// TIA Portal V16 export
// export: Created 2022-11-01T21:54:09.9241492Z, ExportSetting WithDefaults, DisplayName Totally Integrated Automation Portal, DisplayVersion V16, DisplayName TIA Portal Version Control Interface, DisplayVersion V16, DisplayName TIA Portal Openness, DisplayVersion V16, DisplayName SINAMICS Startdrive Advanced, DisplayVersion V16, DisplayName SINAMICS Startdrive G130, G150, S120, S150, SINAMICS MV, S210, DisplayVersion V16, DisplayName SINAMICS Startdrive G110M, G120, G120C, G120D, G120P, DisplayVersion V16, DisplayName STEP 7 Professional, DisplayVersion V16, DisplayName STEP 7 Safety, DisplayVersion V16, DisplayName WinCC Professional, DisplayVersion V16
VAR_GLOBAL   // PLC tag table "AI C700"
   iTIR701 AT %IW1300 : Int;
   iTIR702 AT %IW1302 : Int;
   iTIR703 AT %IW1304 : Int;
   iTIR704 AT %IW1306 : Int;
   iTIR705 AT %IW1308 : Int;
   iTIR706 AT %IW1310 : Int;
   iTIR707 AT %IW1312 : Int;
   iTIR708 AT %IW1314 : Int;
   iTIR709 AT %IW1316 : Int;
   iTIR710 AT %IW1318 : Int;
   iTIR711 AT %IW1320 : Int;
   iTIR712 AT %IW1322 : Int;
   iTIR713 AT %IW1324 : Int;
   iTIR714 AT %IW1326 : Int;
   iTIR715 AT %IW1328 : Int;
   iTIR716 AT %IW1330 : Int;
   iTIR717 AT %IW1332 : Int;
   iTIR718 AT %IW1334 : Int;
   iTIR719 AT %IW1336 : Int;
   iTIR720 AT %IW1338 : Int;
   iTIR721 AT %IW1340 : Int;
   iTIR722 AT %IW1342 : Int;
   iTIR723 AT %IW1344 : Int;
   iTIR724 AT %IW1346 : Int;
   iTIR725 AT %IW1348 : Int;
   iTIR726 AT %IW1350 : Int;
   iTIR727 AT %IW1352 : Int;
   iTIR728 AT %IW1354 : Int;
   iTIR729 AT %IW1356 : Int;
   iTIR730 AT %IW1358 : Int;
   iTIR731 AT %IW1360 : Int;
   iTIR732 AT %IW1362 : Int;
   iTIR733 AT %IW1364 : Int;
   iTIR734 AT %IW1366 : Int;
   iTIR735 AT %IW1368 : Int;
   iTIR736 AT %IW1370 : Int;
   iTIR737 AT %IW1372 : Int;
   iTIR738 AT %IW1374 : Int;
   iTIR739 AT %IW1376 : Int;
   iTIR740 AT %IW1378 : Int;
   iTIR741 AT %IW1380 : Int;
   iTIR742 AT %IW1382 : Int;
   iTIR743 AT %IW1384 : Int;
   iTIR744 AT %IW1386 : Int;
   iTIR745 AT %IW1388 : Int;
   iTIR746 AT %IW1390 : Int;
   iTIR747 AT %IW1392 : Int;
   iTIR748 AT %IW1394 : Int;
   iTIR749 AT %IW1396 : Int;
   iTIR750 AT %IW1398 : Int;
   iTIR751 AT %IW1400 : Int;
   iTIR752 AT %IW1402 : Int;
   iTIR753 AT %IW1404 : Int;
   iTIR754 AT %IW1406 : Int;
   iTIR755 AT %IW1408 : Int;
   iTIR756 AT %IW1410 : Int;
   iTIR757 AT %IW1412 : Int;
   iTIR758 AT %IW1414 : Int;
   iTIR759 AT %IW1416 : Int;
   iTIR760 AT %IW1418 : Int;
   iTIR761 AT %IW1420 : Int;
   iTIR762 AT %IW1422 : Int;
   iQIR701 AT %IW1424 : Int;
   iQIR702 AT %IW1426 : Int;
   iQIR703 AT %IW1428 : Int;
   iQIR704 AT %IW1430 : Int;
   iPIR701 AT %IW1432 : Int;
   iPIR702 AT %IW1434 : Int;
   iPIR703 AT %IW1436 : Int;
   iPIR704 AT %IW1438 : Int;
   iPIR705 AT %IW1440 : Int;
   iPIR706 AT %IW1442 : Int;
   iPIR707 AT %IW1444 : Int;
   iPIR708 AT %IW1446 : Int;
   iPIR709 AT %IW1448 : Int;
   iPIR710 AT %IW1450 : Int;
   iPIR711 AT %IW1452 : Int;
   iPIR712 AT %IW1454 : Int;
   iPIR713_virtual AT %IW1456 : Int;
   iPIR714 AT %IW1458 : Int;
   iPIR715 AT %IW1460 : Int;
   iPIR716_virtual AT %IW1462 : Int;
   iPIR717 AT %IW1464 : Int;
   iPIR718 AT %IW1466 : Int;
   iPIR719_virtual AT %IW1468 : Int;
   iPIR720 AT %IW1470 : Int;
   iPIR721 AT %IW1472 : Int;
   iPIR722 AT %IW1474 : Int;
   iPIR723 AT %IW1476 : Int;
   iPIR724 AT %IW1478 : Int;
   iPIR725 AT %IW1480 : Int;
   iPIR726 AT %IW1482 : Int;
   iPIR727 AT %IW1484 : Int;
   iPIR728 AT %IW1486 : Int;
   iLIR701 AT %IW1488 : Int;
   iLIR702 AT %IW1490 : Int;
   iLIR703 AT %IW1492 : Int;
   iLIR704 AT %IW1494 : Int;
   iLIR705 AT %IW1496 : Int;
   iLIR706 AT %IW1498 : Int;
   iLIR707 AT %IW1500 : Int;
   iLIR708 AT %IW1502 : Int;
   iLIR709 AT %IW1504 : Int;
   iLIR710 AT %IW1506 : Int;
   iLIR711 AT %IW1508 : Int;
   iLIR712 AT %IW1510 : Int;
   iLIR713 AT %IW1512 : Int;
   iLIR714 AT %IW1514 : Int;
   iLIR715 AT %IW1516 : Int;
   iLIR716 AT %IW1518 : Int;
   iLIR717 AT %IW1520 : Int;
   iLIR718 AT %IW1522 : Int;
   iLIR719 AT %IW1524 : Int;
   iLIR720 AT %IW1526 : Int;
   iLIR721 AT %IW1528 : Int;
   iFIR701 AT %IW1530 : Int;
   iFIR702 AT %IW1532 : Int;
   iFIR703 AT %IW1534 : Int;
   iFIR704 AT %IW1536 : Int;
   iFIR705 AT %IW1538 : Int;
   iFIR706 AT %IW1540 : Int;
   iFIR707 AT %IW1542 : Int;
   iFIR708 AT %IW1544 : Int;
   iFIR709 AT %IW1546 : Int;
   iFIR710 AT %IW1548 : Int;
   iFIR711 AT %IW1550 : Int;
   iFIR712 AT %IW1552 : Int;
   iFIR713 AT %IW1554 : Int;
   iFIR714 AT %IW1556 : Int;
   iFIR715 AT %IW1558 : Int;
   iFIR716 AT %IW1560 : Int;
   iFIR717 AT %IW1562 : Int;
   iFIR718 AT %IW1564 : Int;
   iFIR719 AT %IW1566 : Int;
   iFIR720 AT %IW1568 : Int;
   iFIR721 AT %IW1570 : Int;
   iFIR722 AT %IW1572 : Int;
   iFIR723 AT %IW1574 : Int;
   iFIR724 AT %IW1576 : Int;
   iFIR725 AT %IW1578 : Int;
   iFIR726 AT %IW1580 : Int;
   iFIR727 AT %IW1582 : Int;
   iFIR728 AT %IW1584 : Int;
   iLIR722 AT %IW1586 : Int;
END_VAR
